FUNCTION_BLOCK Ob2
VAR_INPUT
END_VAR
VAR_OUTPUT
END_VAR
VAR
	Length : UDINT := 3;
	Height : UDINT := 2;
END_VAR

METHOD Area : UDINT
VAR_INPUT
END_VAR
Area := Length * Height;
END_METHOD

METHOD DefL : UDINT
VAR_INPUT
	L : UDINT;
END_VAR
Length := L;
DefL := Length;
END_METHOD

END_FUNCTION_BLOCK

(* stored: Version 1.1.0.1, ProductVersion 3.1.4018.5
   POU Ob2: Id {2ee00881-c10b-4d2d-8200-a9c948ba3887}, SpecialFunc None
   Method Area: Id {ee34b72b-02b0-4047-b583-1d51441b8d96}
   Method DefL: Id {39c4a7d9-3377-4fe4-9237-47cb10a7412f} *)
